FUNCTION "Trim" : String
TITLE = Trim
{ S7_Optimized_Access := 'TRUE' }
AUTHOR : Machado
FAMILY : 'String'
VERSION : 1.0
//removes leading and trailing whitespace from input string
   VAR_INPUT
      "string" : String;
   END_VAR

   VAR_TEMP
      ret : String;
   END_VAR

   VAR CONSTANT
      space : String := ' ';
   END_VAR


BEGIN
	#ret := #string;
	WHILE LEFT(IN := #ret, L := 1) = #space DO
	    #ret := RIGHT(IN := #ret, L := LEN(#ret) - 1);
	END_WHILE;
	WHILE RIGHT(IN := #ret, L := 1) = #space DO
	    #ret := LEFT(IN := #ret, L := LEN(#ret) - 1);
	END_WHILE;
	#Trim := #ret;
END_FUNCTION

